// TIA Portal V16 export
// export: Created 2022-02-04T14:40:19.3201559Z, ExportSetting WithDefaults, DisplayName Totally Integrated Automation Portal, DisplayVersion V16 Update 1, DisplayName TIA Portal Version Control Interface, DisplayVersion V16, DisplayName TIA Portal Openness, DisplayVersion V16, DisplayName SINAMICS Startdrive Advanced, DisplayVersion V16 Update 5, DisplayName SINAMICS Startdrive G130, G150, S120, S150, SINAMICS MV, S210, DisplayVersion V16 Update 5, DisplayName SINAMICS Startdrive G110M, G120, G120C, G120D, G120P, G115D, DisplayVersion V16 Update 5, DisplayName STEP 7 Professional, DisplayVersion V16, DisplayName STEP 7 Safety, DisplayVersion V16, DisplayName WinCC Advanced, DisplayVersion V16, DisplayName SIMATIC Visualization Architect, DisplayVersion V16
DATA_BLOCK "CNT_CTRL_1"   // DB20
// stored: AutoNumber false, InstanceOfName CNT_CHANTYPE1, OfSystemLibElement CNT_CHANTYPE1, OfSystemLibVersion 1.0
"CNT_CHANTYPE1"
   // VAR RETAIN
   //    AR1_BUFFER : DWord;
   //    FP : Byte;
   //    RESERVED : Byte;
   //    MOD_ADR : Word := 544;
   //    CH_ADR : DWord := P#544.0;
   //    U_D_LGTH : Byte := 16#0;
   //    A_BYTE_0 : Byte;
   //    LOAD_VAL : DInt := 0;
   //    CMP_V1 : DInt;
   //    CMP_V2 : DInt;
   //    A_BIT0_0 : Bool;
   //    TFB : Bool;
   //    A_BIT0_2 : Bool;
   //    A_BIT0_3 : Bool;
   //    A_BIT0_4 : Bool;
   //    A_BIT0_5 : Bool;
   //    A_BIT0_6 : Bool;
   //    A_BIT0_7 : Bool;
   //    ENSET_UP : Bool;
   //    ENSET_DN : Bool;
   //    A_BIT1_2 : Bool;
   //    A_BIT1_3 : Bool;
   //    A_BIT1_4 : Bool;
   //    A_BIT1_5 : Bool;
   //    A_BIT1_6 : Bool;
   //    A_BIT1_7 : Bool;
   //    CTRL_DO0 : Bool;
   //    CTRL_DO1 : Bool;
   //    A_BIT2_2 : Bool;
   //    A_BIT2_3 : Bool;
   //    A_BIT2_4 : Bool;
   //    A_BIT2_5 : Bool;
   //    A_BIT2_6 : Bool;
   //    A_BIT2_7 : Bool;
   //    A_BIT3_0 : Bool;
   //    A_BIT3_1 : Bool;
   //    A_BIT3_2 : Bool;
   //    A_BIT3_3 : Bool;
   //    A_BIT3_4 : Bool;
   //    A_BIT3_5 : Bool;
   //    A_BIT3_6 : Bool;
   //    A_BIT3_7 : Bool;
   //    LATCH_LOAD : DInt;
   //    ACT_CNTV : DInt;
   //    DA_ERR_W : Word;
   //    OT_ERR_B : Byte;
   //    E_BIT0_0 : Bool;
   //    STS_TFB : Bool;
   //    DIAG : Bool;
   //    E_BIT0_3 : Bool;
   //    DATA_ERR : Bool;
   //    E_BIT0_5 : Bool;
   //    E_BIT0_6 : Bool;
   //    PARA : Bool;
   //    E_BYTE_0 : Byte;
   //    STS_RUN : Bool;
   //    STS_DIR : Bool := false;
   //    STS_ZERO : Bool;
   //    STS_OFLW : Bool;
   //    STS_UFLW : Bool;
   //    STS_SYNC : Bool;
   //    STS_GATE : Bool := false;
   //    STS_SW_G : Bool := false;
   //    STS_SET : Bool;
   //    STS_LATCH : Bool;
   //    STS_STA : Bool;
   //    STS_STP : Bool;
   //    STS_CMP1 : Bool;
   //    STS_CMP2 : Bool;
   //    STS_COMP1 : Bool;
   //    STS_COMP2 : Bool;
   //    E_BIT3_0 : Bool;
   //    E_BIT3_1 : Bool;
   //    E_BIT3_2 : Bool;
   //    E_BIT3_3 : Bool;
   //    E_BIT3_4 : Bool;
   //    E_BIT3_5 : Bool;
   //    E_BIT3_6 : Bool;
   //    E_BIT3_7 : Bool;
   //    ACT_CMP1 : DInt;
   //    ACT_CMP2 : DInt;
   //    MDL_DEFECT : Bool;
   //    INT_FAULT : Bool;
   //    EXT_FAULT : Bool;
   //    PNT_INFO : Bool;
   //    EXT_VOLTAGE : Bool;
   //    FLD_CONNCTR : Bool;
   //    NO_CONFIG : Bool;
   //    CONFIG_ERR : Bool;
   //    MDL_TYPE : Byte;
   //    SUB_MDL_ERR : Bool;
   //    COMM_FAULT : Bool;
   //    MDL_STOP : Bool;
   //    WTCH_DOG_FLT : Bool;
   //    INT_PS_FLT : Bool;
   //    PRIM_BATT_FLT : Bool;
   //    BCKUP_BATT_FLT : Bool;
   //    RESERVED_2 : Bool;
   //    RACK_FLT : Bool;
   //    PROC_FLT : Bool;
   //    EPROM_FLT : Bool;
   //    RAM_FLT : Bool;
   //    ADU_FLT : Bool;
   //    FUSE_FLT : Bool;
   //    HW_INTR_FLT : Bool;
   //    RESERVED_3 : Bool;
   //    CH_TYPE : Byte;
   //    LGTH_DIA : Byte;
   //    CH_NO : Byte;
   //    GRP_ERR1 : Bool;
   //    GRP_ERR2 : Bool;
   //    D_BIT7_2 : Bool;
   //    D_BIT7_3 : Bool;
   //    D_BIT7_4 : Bool;
   //    D_BIT7_5 : Bool;
   //    D_BIT7_6 : Bool;
   //    D_BIT7_7 : Bool;
   //    CH1_SIGA : Bool;
   //    CH1_SIGB : Bool;
   //    CH1_SIGZ : Bool;
   //    CH1_BETW : Bool;
   //    CH1_5V2 : Bool;
   //    D_BIT8_5 : Bool;
   //    D_BIT8_6 : Bool;
   //    D_BIT8_7 : Bool;
   //    D_BYTE9 : Byte;
   //    CH2_SIGA : Bool;
   //    CH2_SIGB : Bool;
   //    CH2_SIGZ : Bool;
   //    CH2_BETW : Bool;
   //    CH2_5V2 : Bool;
   //    D_BIT10_5 : Bool;
   //    D_BIT10_6 : Bool;
   //    D_BIT10_7 : Bool;
   //    D_BYTE11 : Byte;
   //    D_BYTE12 : Byte;
   //    D_BYTE13 : Byte;
   //    D_BYTE14 : Byte;
   //    D_BYTE15 : Byte;
   // END_VAR
BEGIN
END_DATA_BLOCK
